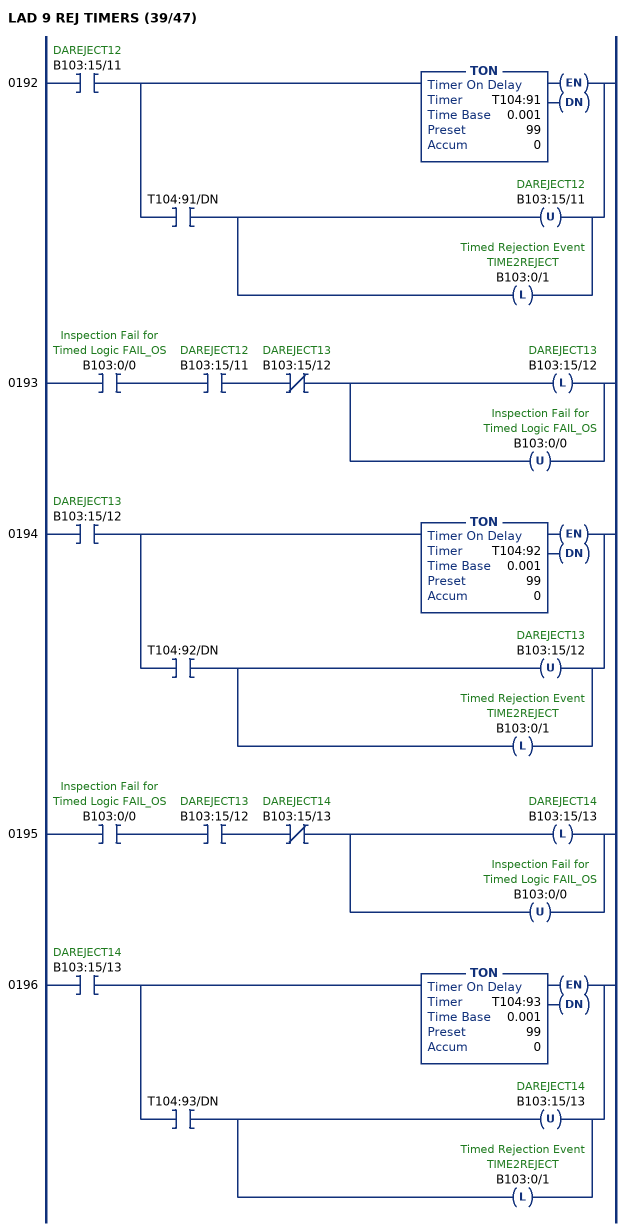
% Rung: 192 %
SOR XIC B103:15/11 BST TON T104:91 0.001 99 0 NXB XIC T104:91/DN BST OTU B103:15/11 NXB OTL B103:0/1 BND BND EOR
%   B103:15/11  DAREJECT12 %
%   B103:0/1  TIME2REJECT  "Timed Rejection Event" %
% Rung: 193 %
SOR XIC B103:0/0 XIC B103:15/11 XIO B103:15/12 BST OTL B103:15/12 NXB OTU B103:0/0 BND EOR
%   B103:0/0  FAIL_OS  "Inspection Fail for Timed Logic" %
%   B103:15/11  DAREJECT12 %
%   B103:15/12  DAREJECT13 %
% Rung: 194 %
SOR XIC B103:15/12 BST TON T104:92 0.001 99 0 NXB XIC T104:92/DN BST OTU B103:15/12 NXB OTL B103:0/1 BND BND EOR
%   B103:15/12  DAREJECT13 %
%   B103:0/1  TIME2REJECT  "Timed Rejection Event" %
% Rung: 195 %
SOR XIC B103:0/0 XIC B103:15/12 XIO B103:15/13 BST OTL B103:15/13 NXB OTU B103:0/0 BND EOR
%   B103:0/0  FAIL_OS  "Inspection Fail for Timed Logic" %
%   B103:15/12  DAREJECT13 %
%   B103:15/13  DAREJECT14 %
% Rung: 196 %
SOR XIC B103:15/13 BST TON T104:93 0.001 99 0 NXB XIC T104:93/DN BST OTU B103:15/13 NXB OTL B103:0/1 BND BND EOR
%   B103:15/13  DAREJECT14 %
%   B103:0/1  TIME2REJECT  "Timed Rejection Event" %

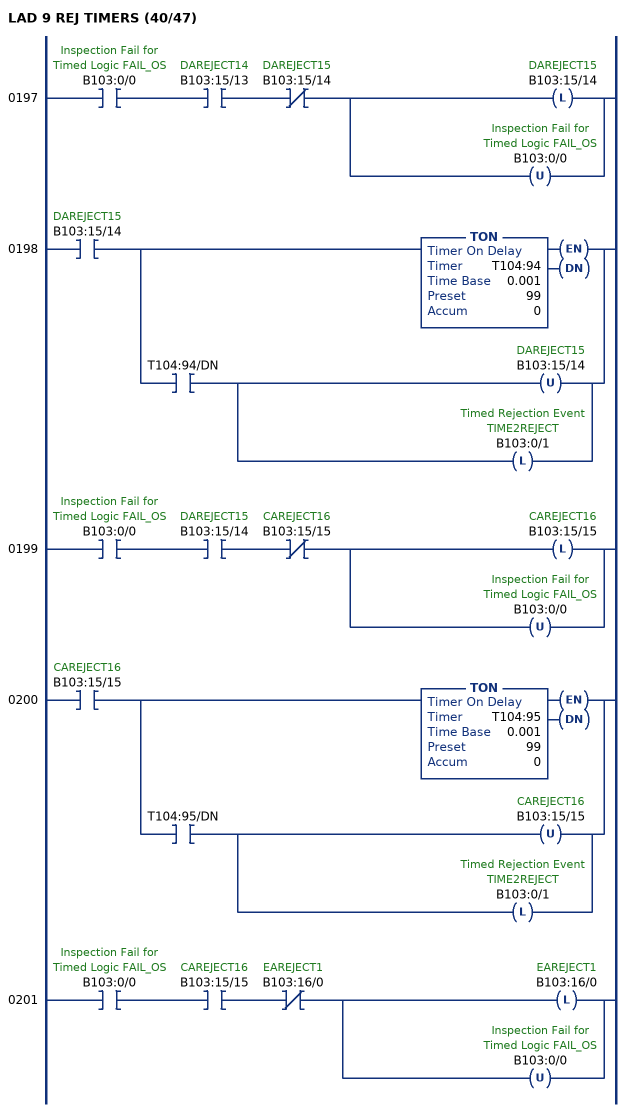
% Rung: 197 %
SOR XIC B103:0/0 XIC B103:15/13 XIO B103:15/14 BST OTL B103:15/14 NXB OTU B103:0/0 BND EOR
%   B103:0/0  FAIL_OS  "Inspection Fail for Timed Logic" %
%   B103:15/13  DAREJECT14 %
%   B103:15/14  DAREJECT15 %
% Rung: 198 %
SOR XIC B103:15/14 BST TON T104:94 0.001 99 0 NXB XIC T104:94/DN BST OTU B103:15/14 NXB OTL B103:0/1 BND BND EOR
%   B103:15/14  DAREJECT15 %
%   B103:0/1  TIME2REJECT  "Timed Rejection Event" %
% Rung: 199 %
SOR XIC B103:0/0 XIC B103:15/14 XIO B103:15/15 BST OTL B103:15/15 NXB OTU B103:0/0 BND EOR
%   B103:0/0  FAIL_OS  "Inspection Fail for Timed Logic" %
%   B103:15/14  DAREJECT15 %
%   B103:15/15  CAREJECT16 %
% Rung: 200 %
SOR XIC B103:15/15 BST TON T104:95 0.001 99 0 NXB XIC T104:95/DN BST OTU B103:15/15 NXB OTL B103:0/1 BND BND EOR
%   B103:15/15  CAREJECT16 %
%   B103:0/1  TIME2REJECT  "Timed Rejection Event" %
% Rung: 201 %
SOR XIC B103:0/0 XIC B103:15/15 XIO B103:16/0 BST OTL B103:16/0 NXB OTU B103:0/0 BND EOR
%   B103:0/0  FAIL_OS  "Inspection Fail for Timed Logic" %
%   B103:15/15  CAREJECT16 %
%   B103:16/0  EAREJECT1 %

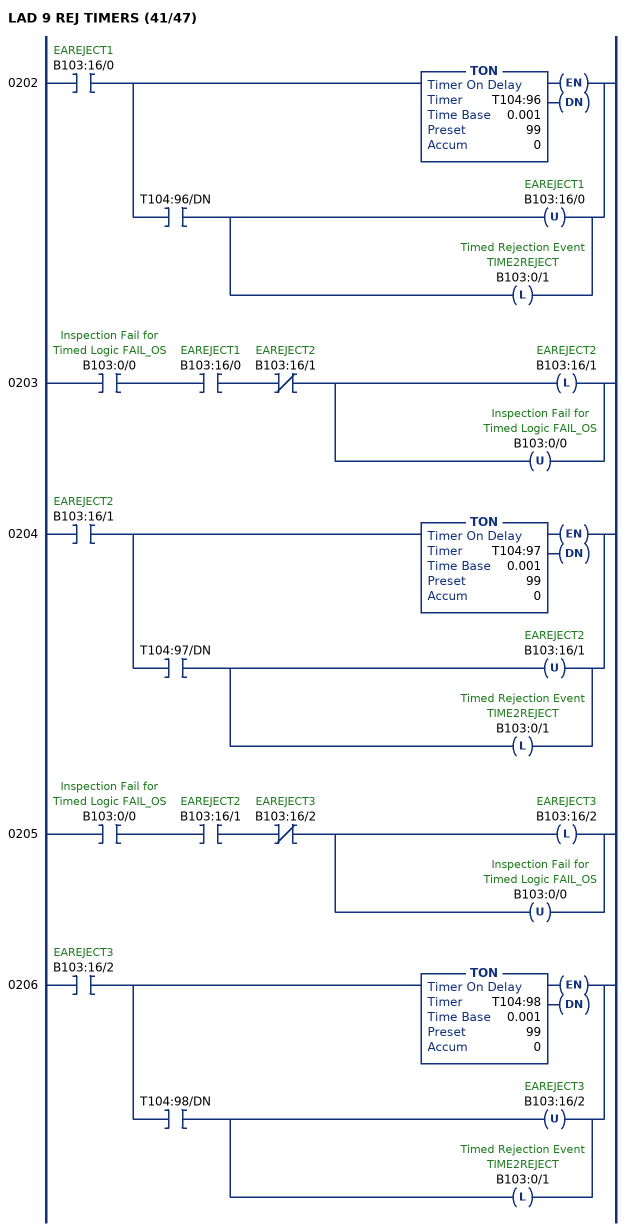
% Rung: 202 %
SOR XIC B103:16/0 BST TON T104:96 0.001 99 0 NXB XIC T104:96/DN BST OTU B103:16/0 NXB OTL B103:0/1 BND BND EOR
%   B103:16/0  EAREJECT1 %
%   B103:0/1  TIME2REJECT  "Timed Rejection Event" %
% Rung: 203 %
SOR XIC B103:0/0 XIC B103:16/0 XIO B103:16/1 BST OTL B103:16/1 NXB OTU B103:0/0 BND EOR
%   B103:0/0  FAIL_OS  "Inspection Fail for Timed Logic" %
%   B103:16/0  EAREJECT1 %
%   B103:16/1  EAREJECT2 %
% Rung: 204 %
SOR XIC B103:16/1 BST TON T104:97 0.001 99 0 NXB XIC T104:97/DN BST OTU B103:16/1 NXB OTL B103:0/1 BND BND EOR
%   B103:16/1  EAREJECT2 %
%   B103:0/1  TIME2REJECT  "Timed Rejection Event" %
% Rung: 205 %
SOR XIC B103:0/0 XIC B103:16/1 XIO B103:16/2 BST OTL B103:16/2 NXB OTU B103:0/0 BND EOR
%   B103:0/0  FAIL_OS  "Inspection Fail for Timed Logic" %
%   B103:16/1  EAREJECT2 %
%   B103:16/2  EAREJECT3 %
% Rung: 206 %
SOR XIC B103:16/2 BST TON T104:98 0.001 99 0 NXB XIC T104:98/DN BST OTU B103:16/2 NXB OTL B103:0/1 BND BND EOR
%   B103:16/2  EAREJECT3 %
%   B103:0/1  TIME2REJECT  "Timed Rejection Event" %

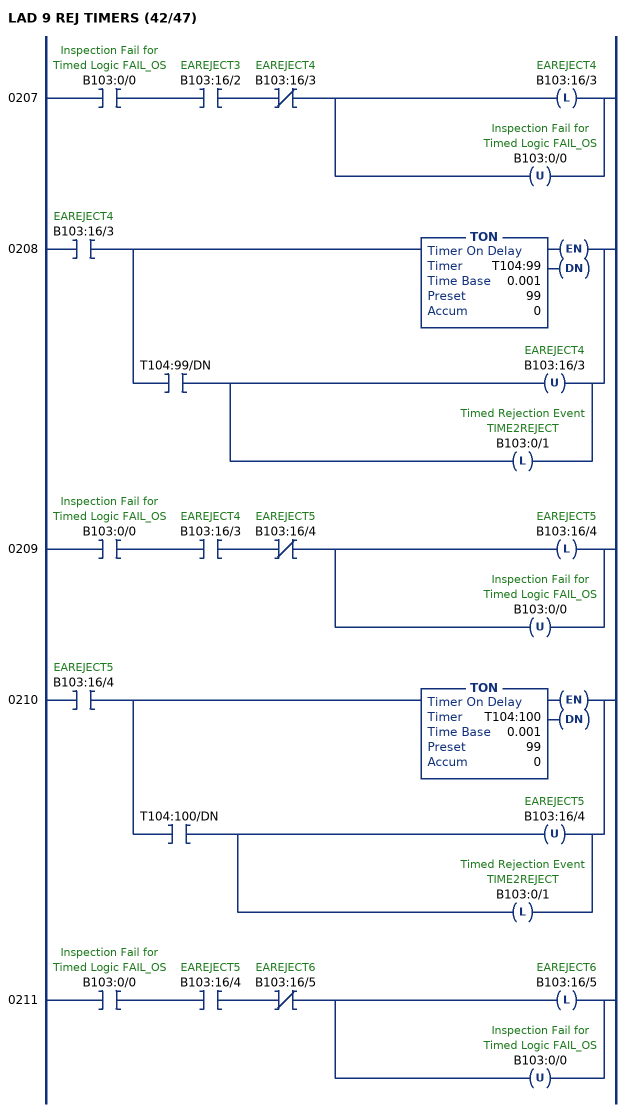
% Rung: 207 %
SOR XIC B103:0/0 XIC B103:16/2 XIO B103:16/3 BST OTL B103:16/3 NXB OTU B103:0/0 BND EOR
%   B103:0/0  FAIL_OS  "Inspection Fail for Timed Logic" %
%   B103:16/2  EAREJECT3 %
%   B103:16/3  EAREJECT4 %
% Rung: 208 %
SOR XIC B103:16/3 BST TON T104:99 0.001 99 0 NXB XIC T104:99/DN BST OTU B103:16/3 NXB OTL B103:0/1 BND BND EOR
%   B103:16/3  EAREJECT4 %
%   B103:0/1  TIME2REJECT  "Timed Rejection Event" %
% Rung: 209 %
SOR XIC B103:0/0 XIC B103:16/3 XIO B103:16/4 BST OTL B103:16/4 NXB OTU B103:0/0 BND EOR
%   B103:0/0  FAIL_OS  "Inspection Fail for Timed Logic" %
%   B103:16/3  EAREJECT4 %
%   B103:16/4  EAREJECT5 %
% Rung: 210 %
SOR XIC B103:16/4 BST TON T104:100 0.001 99 0 NXB XIC T104:100/DN BST OTU B103:16/4 NXB OTL B103:0/1 BND BND EOR
%   B103:16/4  EAREJECT5 %
%   B103:0/1  TIME2REJECT  "Timed Rejection Event" %
% Rung: 211 %
SOR XIC B103:0/0 XIC B103:16/4 XIO B103:16/5 BST OTL B103:16/5 NXB OTU B103:0/0 BND EOR
%   B103:0/0  FAIL_OS  "Inspection Fail for Timed Logic" %
%   B103:16/4  EAREJECT5 %
%   B103:16/5  EAREJECT6 %

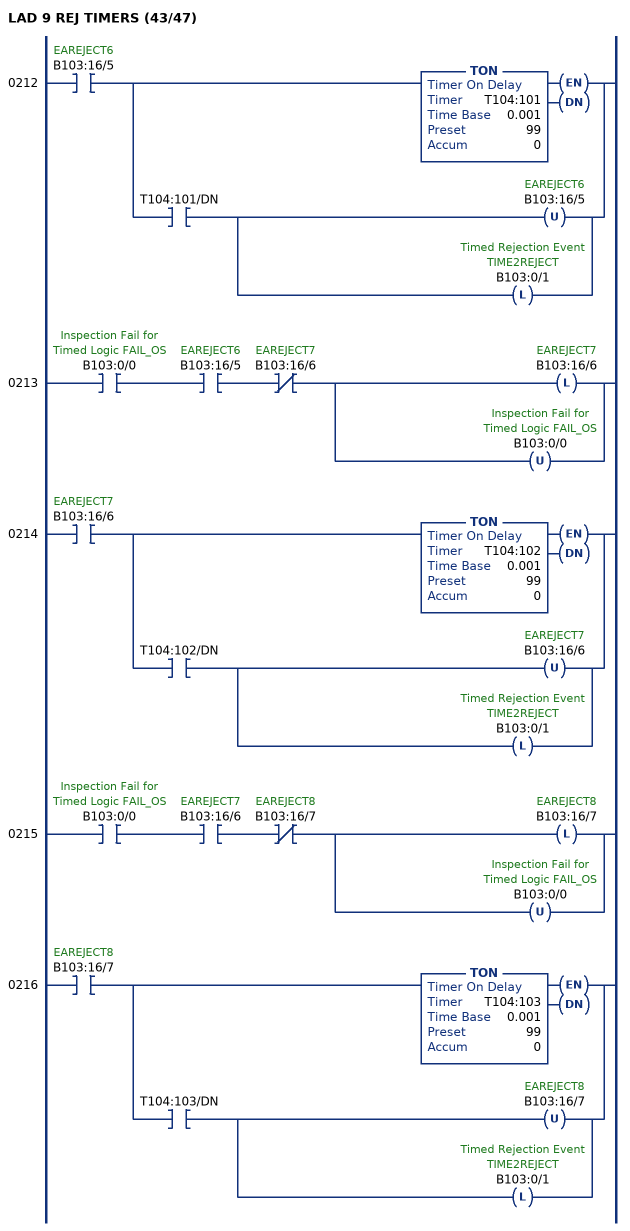
% Rung: 212 %
SOR XIC B103:16/5 BST TON T104:101 0.001 99 0 NXB XIC T104:101/DN BST OTU B103:16/5 NXB OTL B103:0/1 BND BND EOR
%   B103:16/5  EAREJECT6 %
%   B103:0/1  TIME2REJECT  "Timed Rejection Event" %
% Rung: 213 %
SOR XIC B103:0/0 XIC B103:16/5 XIO B103:16/6 BST OTL B103:16/6 NXB OTU B103:0/0 BND EOR
%   B103:0/0  FAIL_OS  "Inspection Fail for Timed Logic" %
%   B103:16/5  EAREJECT6 %
%   B103:16/6  EAREJECT7 %
% Rung: 214 %
SOR XIC B103:16/6 BST TON T104:102 0.001 99 0 NXB XIC T104:102/DN BST OTU B103:16/6 NXB OTL B103:0/1 BND BND EOR
%   B103:16/6  EAREJECT7 %
%   B103:0/1  TIME2REJECT  "Timed Rejection Event" %
% Rung: 215 %
SOR XIC B103:0/0 XIC B103:16/6 XIO B103:16/7 BST OTL B103:16/7 NXB OTU B103:0/0 BND EOR
%   B103:0/0  FAIL_OS  "Inspection Fail for Timed Logic" %
%   B103:16/6  EAREJECT7 %
%   B103:16/7  EAREJECT8 %
% Rung: 216 %
SOR XIC B103:16/7 BST TON T104:103 0.001 99 0 NXB XIC T104:103/DN BST OTU B103:16/7 NXB OTL B103:0/1 BND BND EOR
%   B103:16/7  EAREJECT8 %
%   B103:0/1  TIME2REJECT  "Timed Rejection Event" %

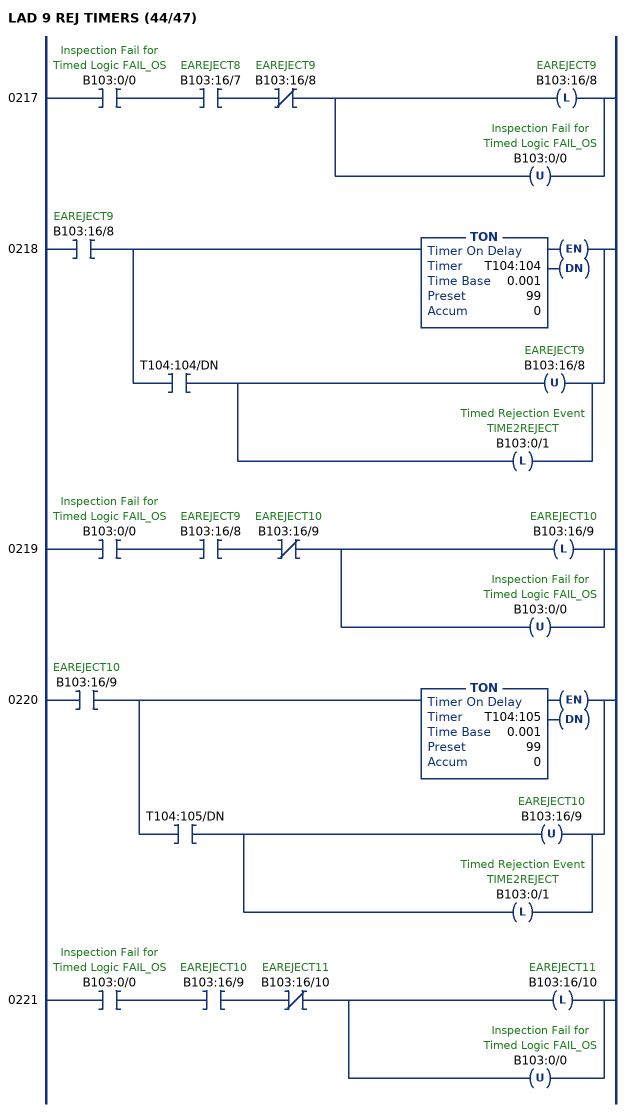
% Rung: 217 %
SOR XIC B103:0/0 XIC B103:16/7 XIO B103:16/8 BST OTL B103:16/8 NXB OTU B103:0/0 BND EOR
%   B103:0/0  FAIL_OS  "Inspection Fail for Timed Logic" %
%   B103:16/7  EAREJECT8 %
%   B103:16/8  EAREJECT9 %
% Rung: 218 %
SOR XIC B103:16/8 BST TON T104:104 0.001 99 0 NXB XIC T104:104/DN BST OTU B103:16/8 NXB OTL B103:0/1 BND BND EOR
%   B103:16/8  EAREJECT9 %
%   B103:0/1  TIME2REJECT  "Timed Rejection Event" %
% Rung: 219 %
SOR XIC B103:0/0 XIC B103:16/8 XIO B103:16/9 BST OTL B103:16/9 NXB OTU B103:0/0 BND EOR
%   B103:0/0  FAIL_OS  "Inspection Fail for Timed Logic" %
%   B103:16/8  EAREJECT9 %
%   B103:16/9  EAREJECT10 %
% Rung: 220 %
SOR XIC B103:16/9 BST TON T104:105 0.001 99 0 NXB XIC T104:105/DN BST OTU B103:16/9 NXB OTL B103:0/1 BND BND EOR
%   B103:16/9  EAREJECT10 %
%   B103:0/1  TIME2REJECT  "Timed Rejection Event" %
% Rung: 221 %
SOR XIC B103:0/0 XIC B103:16/9 XIO B103:16/10 BST OTL B103:16/10 NXB OTU B103:0/0 BND EOR
%   B103:0/0  FAIL_OS  "Inspection Fail for Timed Logic" %
%   B103:16/9  EAREJECT10 %
%   B103:16/10  EAREJECT11 %

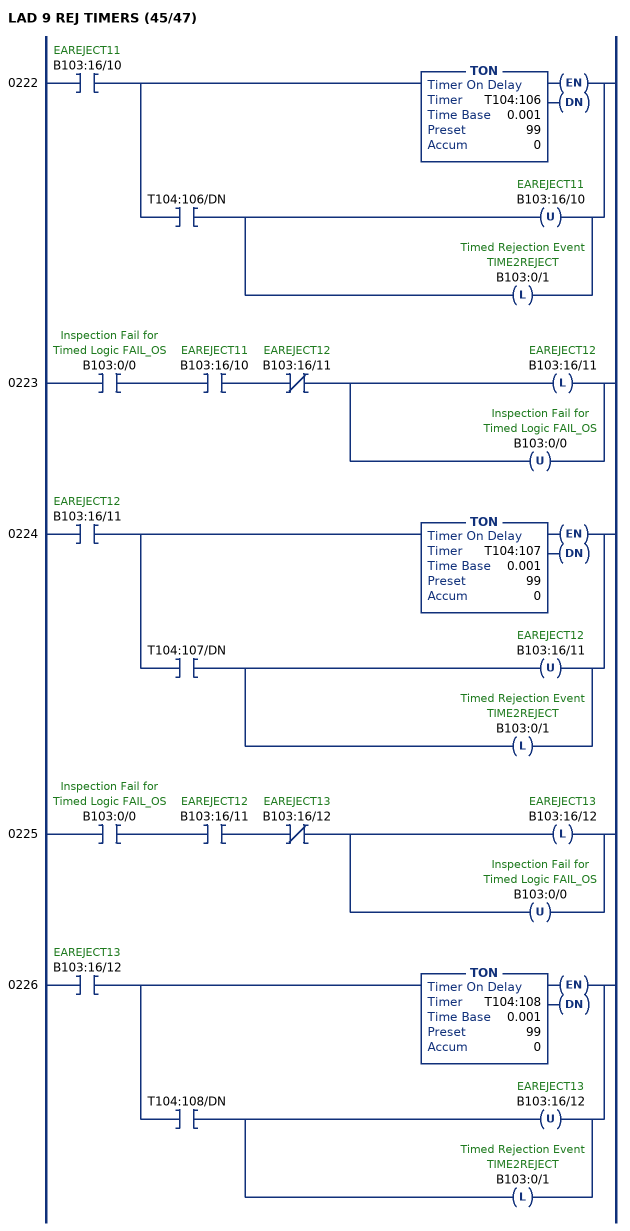
% Rung: 222 %
SOR XIC B103:16/10 BST TON T104:106 0.001 99 0 NXB XIC T104:106/DN BST OTU B103:16/10 NXB OTL B103:0/1 BND BND EOR
%   B103:16/10  EAREJECT11 %
%   B103:0/1  TIME2REJECT  "Timed Rejection Event" %
% Rung: 223 %
SOR XIC B103:0/0 XIC B103:16/10 XIO B103:16/11 BST OTL B103:16/11 NXB OTU B103:0/0 BND EOR
%   B103:0/0  FAIL_OS  "Inspection Fail for Timed Logic" %
%   B103:16/10  EAREJECT11 %
%   B103:16/11  EAREJECT12 %
% Rung: 224 %
SOR XIC B103:16/11 BST TON T104:107 0.001 99 0 NXB XIC T104:107/DN BST OTU B103:16/11 NXB OTL B103:0/1 BND BND EOR
%   B103:16/11  EAREJECT12 %
%   B103:0/1  TIME2REJECT  "Timed Rejection Event" %
% Rung: 225 %
SOR XIC B103:0/0 XIC B103:16/11 XIO B103:16/12 BST OTL B103:16/12 NXB OTU B103:0/0 BND EOR
%   B103:0/0  FAIL_OS  "Inspection Fail for Timed Logic" %
%   B103:16/11  EAREJECT12 %
%   B103:16/12  EAREJECT13 %
% Rung: 226 %
SOR XIC B103:16/12 BST TON T104:108 0.001 99 0 NXB XIC T104:108/DN BST OTU B103:16/12 NXB OTL B103:0/1 BND BND EOR
%   B103:16/12  EAREJECT13 %
%   B103:0/1  TIME2REJECT  "Timed Rejection Event" %

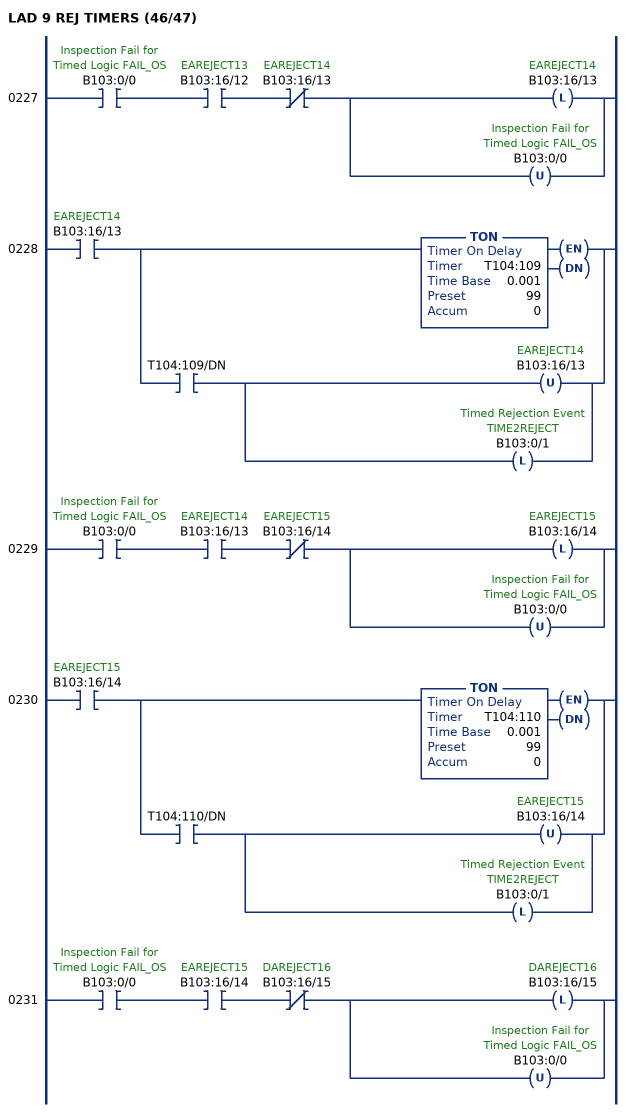
% Rung: 227 %
SOR XIC B103:0/0 XIC B103:16/12 XIO B103:16/13 BST OTL B103:16/13 NXB OTU B103:0/0 BND EOR
%   B103:0/0  FAIL_OS  "Inspection Fail for Timed Logic" %
%   B103:16/12  EAREJECT13 %
%   B103:16/13  EAREJECT14 %
% Rung: 228 %
SOR XIC B103:16/13 BST TON T104:109 0.001 99 0 NXB XIC T104:109/DN BST OTU B103:16/13 NXB OTL B103:0/1 BND BND EOR
%   B103:16/13  EAREJECT14 %
%   B103:0/1  TIME2REJECT  "Timed Rejection Event" %
% Rung: 229 %
SOR XIC B103:0/0 XIC B103:16/13 XIO B103:16/14 BST OTL B103:16/14 NXB OTU B103:0/0 BND EOR
%   B103:0/0  FAIL_OS  "Inspection Fail for Timed Logic" %
%   B103:16/13  EAREJECT14 %
%   B103:16/14  EAREJECT15 %
% Rung: 230 %
SOR XIC B103:16/14 BST TON T104:110 0.001 99 0 NXB XIC T104:110/DN BST OTU B103:16/14 NXB OTL B103:0/1 BND BND EOR
%   B103:16/14  EAREJECT15 %
%   B103:0/1  TIME2REJECT  "Timed Rejection Event" %
% Rung: 231 %
SOR XIC B103:0/0 XIC B103:16/14 XIO B103:16/15 BST OTL B103:16/15 NXB OTU B103:0/0 BND EOR
%   B103:0/0  FAIL_OS  "Inspection Fail for Timed Logic" %
%   B103:16/14  EAREJECT15 %
%   B103:16/15  DAREJECT16 %

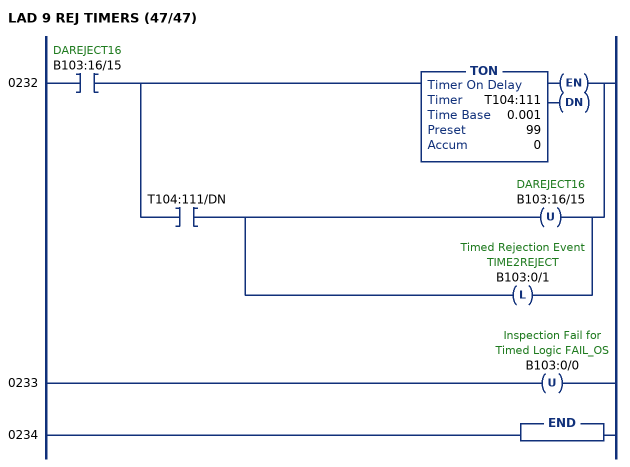
% Rung: 232 %
SOR XIC B103:16/15 BST TON T104:111 0.001 99 0 NXB XIC T104:111/DN BST OTU B103:16/15 NXB OTL B103:0/1 BND BND EOR
%   B103:16/15  DAREJECT16 %
%   B103:0/1  TIME2REJECT  "Timed Rejection Event" %
% Rung: 233 %
SOR OTU B103:0/0 EOR
%   B103:0/0  FAIL_OS  "Inspection Fail for Timed Logic" %
% Rung: 234 %
SOR END EOR

LADDER 10 "1MS_SCAN"
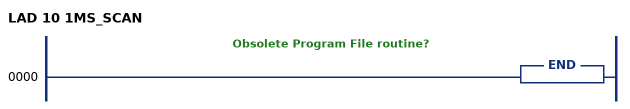
% Rung: 0 %
% TITLE: Obsolete Program File routine? %
SOR END EOR

LADDER 11 "HSC0"
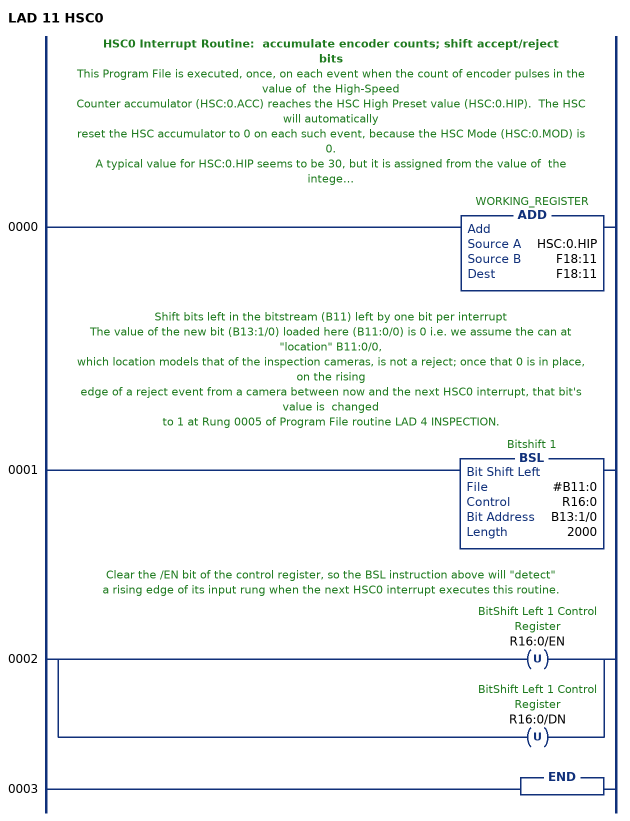
% Rung: 0 %
% TITLE: HSC0 Interrupt Routine:  accumulate encoder counts; shift accept/reject bits %
% This Program File is executed, once, on each event when the count of encoder pulses in the value of  the High-Speed
% Counter accumulator (HSC:0.ACC) reaches the HSC High Preset value (HSC:0.HIP).  The HSC will automatically
% reset the HSC accumulator to 0 on each such event, because the HSC Mode (HSC:0.MOD) is 0.
% 
% A typical value for HSC:0.HIP seems to be 30, but it is assigned from the value of  the integer
% ENCODER_HIPRESET_SP (N7:11) in the INSPECTION routine (LAD 4)  at Rung 0002. whenever
% 
%   1) the bit USE_ENCODER (B3:0/11) is 1, and
%   2) ENCODER_HIPRESET_SP differs from HSC:0.HIP.
% 
% Both USE_ENCODER and ENCODER_HIPRESET_SP originate in the GUI HMI..
% 
% The HSC function is only enabled (HSC:0/FE) when USE_ENCODER is 1,
% per the assignment of HSC:0/FE in MAIN_PROG routine (LAD 2) Rung 0002.
% 
% ========================================================================
% 
% Rung 0000 adds the HSC High Preset value to the value of a working register, which register
% will, at regular intervals (300ms)*, be
% 
%   1) Scaled to estimate the line speed, and
%   2) Cleared to 0.0 to initialize the estimate for the next interval
% 
% * Program File routine LAD 13 STI_SPEED, via Selectable Timed Interrupt %
SOR ADD HSC:0.HIP F18:11 F18:11 EOR
%   F18:11  WORKING_REGISTER %
% Rung: 1 %
% Shift bits left in the bitstream (B11) left by one bit per interrupt
% 
% The value of the new bit (B13:1/0) loaded here (B11:0/0) is 0 i.e. we assume the can at "location" B11:0/0,
% which location models that of the inspection cameras, is not a reject; once that 0 is in place, on the rising
% edge of a reject event from a camera between now and the next HSC0 interrupt, that bit's value is  changed
% to 1 at Rung 0005 of Program File routine LAD 4 INSPECTION. %
SOR BSL #B11:0 R16:0 B13:1/0 2000 EOR
%   B11:0  "Bitshift 1" %
%   R16:0  "BitShift Left 1 Control Register" %
%   B13:1/0  "BSL Load point (unused placeholder)" %
% Rung: 2 %
% Clear the /EN bit of the control register, so the BSL instruction above will "detect"
% a rising edge of its input rung when the next HSC0 interrupt executes this routine. %
SOR BST OTU R16:0/EN NXB OTU R16:0/DN BND EOR
%   R16:0  "BitShift Left 1 Control Register" %
% Rung: 3 %
SOR END EOR

LADDER 12 "EII_COUNTS"    % count events to determine speed %
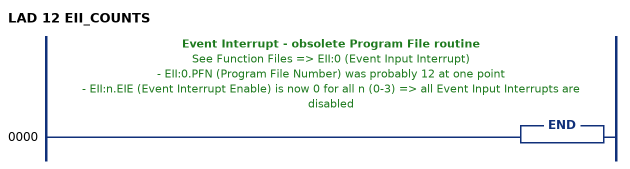
% Rung: 0 %
% TITLE: Event Interrupt - obsolete Program File routine %
% See Function Files => EII:0 (Event Input Interrupt)
% 
% - EII:0.PFN (Program File Number) was probably 12 at one point
% - EII:n.EIE (Event Interrupt Enable) is now 0 for all n (0-3) => all Event Input Interrupts are disabled %
SOR END EOR

LADDER 13 "STI_SPEED"    % calc line speed based on eii counts %
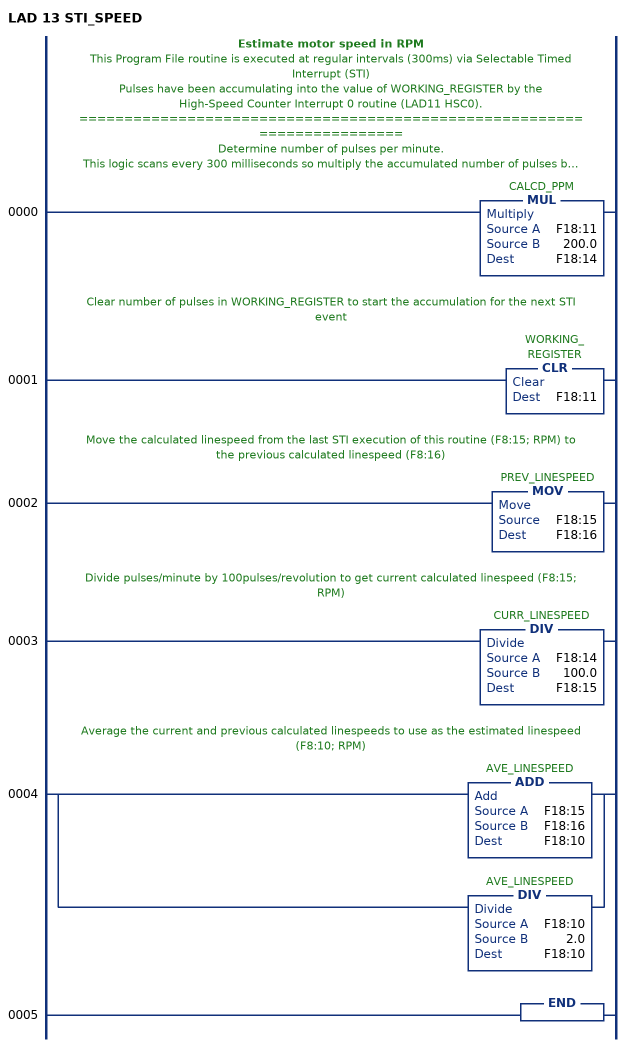
% Rung: 0 %
% TITLE: Estimate motor speed in RPM %
% This Program File routine is executed at regular intervals (300ms) via Selectable Timed Interrupt (STI)
% 
% Pulses have been accumulating into the value of WORKING_REGISTER by the
% High-Speed Counter Interrupt 0 routine (LAD11 HSC0).
% 
% ========================================================================
% Determine number of pulses per minute.
% This logic scans every 300 milliseconds so multiply the accumulated number of pulses by 200
% to calculate the number of pulses per minute %
SOR MUL F18:11 200.0 F18:14 EOR
%   F18:11  WORKING_REGISTER %
%   F18:14  CALCD_PPM %
% Rung: 1 %
% Clear number of pulses in WORKING_REGISTER to start the accumulation for the next STI event %
SOR CLR F18:11 EOR
%   F18:11  WORKING_REGISTER %
% Rung: 2 %
% Move the calculated linespeed from the last STI execution of this routine (F8:15; RPM) to the previous calculated linespeed (F8:16) %
SOR MOV F18:15 F18:16 EOR
%   F18:15  "CURR_LINESPEED" %
%   F18:16  PREV_LINESPEED %
% Rung: 3 %
% Divide pulses/minute by 100pulses/revolution to get current calculated linespeed (F8:15; RPM) %
SOR DIV F18:14 100.0 F18:15 EOR
%   F18:14  CALCD_PPM %
%   F18:15  "CURR_LINESPEED" %
% Rung: 4 %
% Average the current and previous calculated linespeeds to use as the estimated linespeed (F8:10; RPM) %
SOR BST ADD F18:15 F18:16 F18:10 NXB DIV F18:10 2.0 F18:10 BND EOR
%   F18:15  "CURR_LINESPEED" %
%   F18:16  PREV_LINESPEED %
%   F18:10  AVE_LINESPEED %
% Rung: 5 %
SOR END EOR

OTHER DOCUMENTED ADDRESSES
  B3:0/1  "update rejection timer duration"
  B3:0/7  NOP
  B3:0/9  UPDATETIMERS
  B3:1/2  "Red Light ON-Caser"
  B3:1/3  "Consecutive Rejects Stop Can Code"
  B3:1/4  "Red Light ON"
  B3:1/5  "Red Light OFF Bit"
  B3:1/6  "Consecutive Rehjects Stop Labeler Machine"
  B3:1/7  "Red Light On-Labeler"
  B3:1/8  "Red Light Off Bit"
  B3:1/9  "Red Light OFF Bit"
  B3:1/10  "Red Light ON Manual Activate"
  B3:2/14  "Can Code Consecutive Rejects Bit"
  B3:2/15  "VAriety Code Consecutive Rejects Bit"
  B3:3/0  "RESET PB From VB Application"
  B3:3/1  "One Shot"
  B13:0/0  HEARTBEAT_FROM_GUI
  B13:1/1  "Commit new HSC0 values"
  B13:1/8  "Inspection Mode: ERROR"
  B13:1/9  "Inspection Mode: OFF (Disabled)"
  B13:1/10  "Inspection Mode: TESTING (rejection and Linestop disabled for period of time)"
  B13:1/11  "Inspection Mode: ACTIVE (Enabled)"
  B13:2/2  A_ONESHOT2
  B13:5  INSPECTION_SEQ
  B13:5/0  TRIGGERED
  B13:5/2  PASS_RESULT
  B13:8/0  "OutTest0"
  B13:8/1  "OutTest1"
  B13:9/0  "ONS Test 0"
  B21:0  "Bitshift 2"
  B23:0/15  "Labeler Reject Commmand"
  B23:1/0  "BSL Load point"
  B23:1/1  "Labeler Commit new HSC1 values"
  B23:1/8  "Labeler Vision System ERROR/FAULT"
  B23:1/9  "Labeler Vision System INACTIVE"
  B23:1/10  "Labeler Vision System TESTING (rejection and Linestop disabled for period of time)"
  B23:1/11  "Labeler Vision System ACTIVE"
  B23:2/0  B_ONESHOT0
  B23:2/1  B_ONESHOT1
  B23:2/2  B_ONESHOT2
  B33:1/8  "Caser BarCode Vision System ERROR/FAULT"
  B33:1/9  "Caser BarCode Vision System INACTIVE"
  B33:1/10  "Caser BarCode Vision System TESTING (rejection and Linestop disabled for period of time)"
  B33:1/11  "Caser BarCode Vision System ACTIVE"
  DFILE:0  "OUTPUT"
  DFILE:1  "INPUT"
  DFILE:2  "STATUS"
  DFILE:3  "BINARY"
  DFILE:4  "TIMER"
  DFILE:5  "COUNTER"
  DFILE:6  "CONTROL"
  DFILE:7  "INTEGER"
  DFILE:8  "FLOAT"
  DFILE:10  "WORKBITS1"
  DFILE:11  "BITSHIFT1"
  DFILE:13  "WORKBITS1"
  DFILE:14  "TIMERS1"
  DFILE:15  "COUNTERS1"
  DFILE:16  "CTRLREGS1"
  DFILE:17  "INTEGERS1"
  DFILE:18  "FLOATS1"
  DFILE:20  "CONS REJEC"
  DFILE:21  "BITSHIFT2"
  DFILE:23  "WORKBITS2"
  DFILE:24  "TIMERS2"
  DFILE:25  "COUNTERS2"
  DFILE:26  "CTRLREGS2"
  DFILE:27  "INTEGERS2"
  DFILE:93  "TEMP BITS just in case"
  DFILE:94  "TEMP TMRS just in case"
  DFILE:95  "TEMP CTRS just in case"
  DFILE:96  "TEMP CTRL just in case"
  DFILE:97  "TEMP INTS just in case"
  DFILE:98  "TEMP FLTS just in case"
  DFILE:99  "RIX"
  DFILE:100  "MSG"
  DFILE:103  "TIMEDBITS Bits used for 100 ti med rejections"
  DFILE:104  "TIMEDTMRS Timers used for 100 timed rejections"
  EII:0.0  "call program file 12"
  EII:0.2/14  "1 = rising edge"
  EII:0.3  "2 = input 2"
  ES1:5/0  PLC_COMM_TOPC_OK
  F18:0  TOTAL_INSPECTED_GUI  "Total Inspected Count from GUI"
  F18:1  TOTAL_PASSED_GUI  "Total Passed Count from GUI"
  F18:2  TOTAL_FAILED_GUI  "Total Failed Count from GUI"
  F18:3  TOTAL_REJECTED_GUI  "Total Reject Count from GUI"
  F18:17  LOWSPEED_RPM_SP
  HSC:0  "Inspection Code Bitshift"
  HSC:0.3/15  "Encoder Count Event"
  HSC:0.5  "Each time .HIP is reached it shifts bitstream"
  HSC:0.7  "HSC:0 HI PRESET"
  HSC:1  "Labeler Bitshift"
  HSC:1.5  "Each time .HIP is reached it shifts bitstream"
  HSC:1.7  "HSC:1 HI PRESET"
  HSC:3  "Variety LineSpeed"
  I:0.0/0  HSC_ENCODER  "Encoder Input"
  N7:4/6  CASE2_RED
  N20:1  "Consecutive Rejects From Labeler"
  N21:0  "Reset PB From VB Application, Sends a 1 to N21:0"
  N22:0  "RESET PB from VB Application; Seta a 1 to N22:0"
  N27:0  "Labeler Vision Inspection Mode ERROR, INACTIVE, TESTING, ACTIVE"
  N27:1  "Labeler Reject Offset (HSC increments from camera result area)"
  N27:6  "Linestop Triggered from VB"
  N37:0  "Caser BarCode Inspection ERROR, INACTIVE, TESTING, ACTIVE"
  N37:6  "Linestop Triggered from VB"
  Q9:1  LOOP_120_TIMES
  R26:0  "BitShift Left 2 Control Register"
  ST19:0  PLC_REVISION  "PLC REVISION Displayed on GUI"
  ST19:1  CURRENT_JOBFILE  "CURRENT JOB from GUI"
  ST19:2  CURRENT_OPERATOR  "Current Operator Logged In from GUI"
  T24:0  "Seamer B Reject Actuator Dwell Timer"
  T24:0.PRE  "<-- should be 50 at a minimum"
  U:6  "CASER CODE LOGIC"

COMMENTS NOT ATTACHED TO A CURRENT RUNG
  N17:5: The ADJUSTED_OFFSET is the bit position where the rejection should occur.  Because it is used as an indirect reference in the ladder logic, this must be an integer so the calulated value is cast to an integer value to drop fractional parts.
  F18:2: offset calculation is                              ( OFFSET AT FASTEST [N17:3] + (CALCD RPM [F18:0]  - MAX RPM [F18:8] )  multilied by slope (below)
    
    
    slope =                                         ( OFFSET AT FASTEST [ N17:3] - OFFSET AT SLOWEST [N17:1] ) /  ( MAX RPM [F18:8] - MIN RPM [F18:7] )
  F18:0: For Markesan: Can Code Linespeed range is 20 to 40 so at its lowest speed (20) the encoder counts 1556 pulses.  This is used to calculate line speed which is then used to advance/retard the rejection timing between the two offset setpoints.  Multiply this value times 30 to calculate the number of pulses per minute.
  B23:1/8: Seamer Mode Status from Vision System
  B23:1/1: ============================================================================================
    To commit the HSC parameters, change the value of Hi Preset (N7:0) and/or Lo Preset (N7:1) then set bit B23:1/1.
    This HSL will load the new parameters into the HSC subsystem then the bit will unlatch (reset).
    ============================================================================================
  B23:0/15: Rejection Logic / ============================================================================================
    The bitshift conveys the fail status from the point of origin each time the HSC Hi Preset is reached.  The REJECT output should fire at a point in the future as assigned by the value of N27:1 which is changeable in the data table.  Once this REJECT signal is set, it should be tied to the actual output to trigger the reject actuator then this bit should be reset once kickout has fired.
    ============================================================================================
  B21:0: ============================================================================================
    This subroutine fires each time HSC0 accumulated counts meets the HI or LO preset.  Since we do not care (and should never get a LO, this logic executes a bitshift.  If the bits are shifted too much, increas the HI preset.  It is suggested that we get close to 10 shifts per can, the better "resolution" the better the kickout accuracy.  Please remember that varied latency in the assignment of the PASS or FAIL result may place this status in inconsistent locations of the bitshift so resolution must be adequate for that but noot too fine as to be shift intensive.
    ============================================================================================
  B13:1/8: Variety Code Mode Status from Vision System
  B13:1/1: ============================================================================================
    To commit the HSC parameters, change the value of Hi Preset (N7:0) and/or Lo Preset (N7:1) then set bit B13:1/1.
    This HSL will load the new parameters into the HSC subsystem then the bit will unlatch (reset).
    ============================================================================================

REVISION NOTES
  0: Moving Inputs to new config

DATA TABLE (non-zero values as saved)
DATA B3
% B3:0 % 0X8048 0X0008 0X0007 0X0008 0X0000
DATA T4
% .PRE .ACC %
% T4:0 % 500 0
% T4:1 % 3 0
% T4:2 % 1 0
% T4:3 % 1 0
% T4:4 % 1 0
% T4:5 % 1 0
% T4:6 % 1 0
% T4:7 % 1 0
% T4:8 % 1 0
% T4:9 % 1 0
% T4:10 % 1 0
% T4:11 % 1 0
% T4:12 % 1 0
% T4:13 % 40 0
% T4:14 % 15 0
% T4:15 % 40 0
% T4:16 % 15 0
% T4:17 % 40 0
% T4:18 % 15 0
% T4:19 % 1 0
% T4:20 % 50 50
% T4:21 % 1 0
% T4:22 % 50 0
% T4:23 % 32767 130
DATA C5
% .PRE .ACC %
% C5:1 % 0 -32737
% C5:2 % 0 348
% C5:9 % 112 112
DATA N7
% N7:0 % 10 10 0 0 0 0 0 0 0 0
% N7:10 % 1 3 0 0 0 0 0 0 0 0
% N7:20 % 500 0 0 0 0 0 0 0 0 0
DATA F8
% F8:0 % 17640 0
DATA B11
% B11:0 % 0X0001 0X0000 0X0000 0X0000 0X0000 0X0000 0X0000 0X0000 0X0000 0X0000
% B11:20 % 0X0000 0X0000 0X0000 0X0000 0X0000 0X0000 0X0000 0X0000 0X0000 0X2000
% B11:50 % 0X0000 0X0000 0X0000 0X0000 0X0000 0X0000 0X0020 0X0000 0X0000 0X0000
% B11:70 % 0X0000 0X0000 0X0000 0X0000 0X0000 0X0000 0X0000 0X0000 0X0000 0X0008
% B11:100 % 0X0000 0X0001 0X0000 0X0000 0X0000 0X0000 0X0000 0X0000 0X0000 0X0000
DATA B13
% B13:0 % 0X0001 0X0000 0X0000 0X00FF 0X0000 0X0000 0X0000 0X0000 0X0000 0X0000
DATA T14
% .PRE .ACC %
% T14:0 % 55 0
% T14:2 % 70 0
% T14:3 % 1 0
% T14:5 % 1 0
% T14:6 % 3 3
% T14:7 % 3 3
% T14:8 % 5 0
% T14:9 % 50 0
DATA C15
% .PRE .ACC %
% C15:0 % 0 -32756
% C15:1 % 0 951
DATA R16
% .LEN .POS %
% R16:0 % 2000 0
DATA N17
% N17:0 % 1000 250 0 0 0 55 0 0 0 0
% N17:10 % 0 30
DATA F18
% F18:0 % 38 38 0 0 0
% F18:10 % 0 0 250 0 0
% F18:15 % 0 0 0 710 0
% F18:30 % 0 0 -750 0 0
DATA ST19
% ST19:0 % "2023-01-13"
% ST19:1 % "C:\Tensor\TensorVisionZ\Code\Zebra\Aurora\TwoCam1.avproj"
% ST19:2 % "TensorID"
DATA T104
% .PRE .ACC %
% T104:0 % 9 0
% T104:1 % 9 0
% T104:2 % 9 0
% T104:3 % 9 0
% T104:4 % 9 0
% T104:5 % 9 0
% T104:6 % 9 0
% T104:7 % 9 0
% T104:8 % 9 0
% T104:9 % 9 0
% T104:10 % 9 0
% T104:11 % 9 0
% T104:12 % 9 0
% T104:13 % 9 0
% T104:14 % 9 0
% T104:15 % 9 0
% T104:16 % 9 0
% T104:17 % 9 0
% T104:18 % 9 0
% T104:19 % 9 0
% T104:20 % 9 0
% T104:21 % 9 0
% T104:22 % 9 0
% T104:23 % 9 0
% T104:24 % 9 0
% T104:25 % 9 0
% T104:26 % 9 0
% T104:27 % 9 0
% T104:28 % 9 0
% T104:29 % 9 0
% T104:30 % 9 0
% T104:31 % 9 0
% T104:32 % 9 0
% T104:33 % 9 0
% T104:34 % 9 0
% T104:35 % 9 0
% T104:36 % 9 0
% T104:37 % 9 0
% T104:38 % 9 0
% T104:39 % 9 0
% T104:40 % 9 0
% T104:41 % 9 0
% T104:42 % 9 0
% T104:43 % 9 0
% T104:44 % 9 0
% T104:45 % 9 0
% T104:46 % 9 0
% T104:47 % 9 0
% T104:48 % 9 0
% T104:49 % 9 0
% T104:50 % 99 0
% T104:51 % 99 0
% T104:52 % 99 0
% T104:53 % 99 0
% T104:54 % 9 0
% T104:55 % 9 0
% T104:56 % 9 0
% T104:57 % 9 0
% T104:58 % 9 0
% T104:59 % 9 0
% T104:60 % 9 0
% T104:61 % 9 0
% T104:62 % 99 0
% T104:63 % 99 0
% T104:64 % 99 0
% T104:65 % 99 0
% T104:66 % 99 0
% T104:67 % 99 0
% T104:68 % 99 0
% T104:69 % 99 0
% T104:70 % 99 0
% T104:71 % 99 0
% T104:72 % 99 0
% T104:73 % 99 0
% T104:74 % 99 0
% T104:75 % 99 0
% T104:76 % 99 0
% T104:77 % 99 0
% T104:78 % 99 0
% T104:79 % 99 0
% T104:80 % 99 0
% T104:81 % 99 0
% T104:82 % 99 0
% T104:83 % 99 0
% T104:84 % 99 0
% T104:85 % 99 0
% T104:86 % 99 0
% T104:87 % 99 0
% T104:88 % 99 0
% T104:89 % 99 0
% T104:90 % 99 0
% T104:91 % 99 0
% T104:92 % 99 0
% T104:93 % 99 0
% T104:94 % 99 0
% T104:95 % 99 0
% T104:96 % 99 0
% T104:97 % 99 0
% T104:98 % 99 0
% T104:99 % 99 0
% T104:100 % 99 0
% T104:101 % 99 0
% T104:102 % 99 0
% T104:103 % 99 0
% T104:104 % 99 0
% T104:105 % 99 0
% T104:106 % 99 0
% T104:107 % 99 0
% T104:108 % 99 0
% T104:109 % 99 0
% T104:110 % 99 0
% T104:111 % 99 0
% T104:112 % 250 0
% T104:113 % 295 0
% T104:114 % 295 0
